FUNCTION_BLOCK Assignment
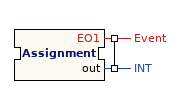
  EVENT_OUTPUT
    EO1 WITH out;
  END_EVENT
  VAR_OUTPUT
    out : INT;
  END_VAR
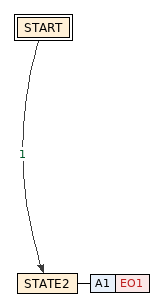
  EC_STATES
    START;
    STATE2 : A1 -> EO1;
  END_STATES
  EC_TRANSITIONS
    START TO STATE2 := 1;
  END_TRANSITIONS
  ALGORITHM A1 IN ST:
  VAR_TEMP
    t : INT;
  END_VAR
t := 6;&#38;#10;out := 4;&#38;#10;
  END_ALGORITHM
END_FUNCTION_BLOCK
